// TIA Portal V19 export
TYPE "LEXCHANGETRAY_typeRollerIoSignalManualCommands_B2"
// trayAutomaticFeedingDetectionU2Em6: Bool
// stored: Access Published
   STRUCT
      trayAutomaticFeedingDetectionU2Em6 : Bool;
   END_STRUCT;
END_TYPE
